PROGRAM PRG_Compilation
VAR
END_VAR

END_PROGRAM

(* stored: Version 1.1.0.1
   POU PRG_Compilation: Id {b1995b4c-786d-03c5-204c-1db0d16f2c14}, SpecialFunc None *)
